TYPE ST_MainAxisInterface :
STRUCT
	stMainAxisInterface_stat		: ST_MainAxisInterface_Stat;
	stMainAxisInterface_ctrl		: ST_MainAxisInterface_Ctrl;
END_STRUCT
END_TYPE

(* stored: Version 1.1.0.1, ProductVersion 3.1.4024.12
   DUT ST_MainAxisInterface: Id {f5f66309-d347-497a-b131-c96e2eb2505f} *)
